RoboDK station: Stringer B Corner-Top-Short-BOX1.rdk

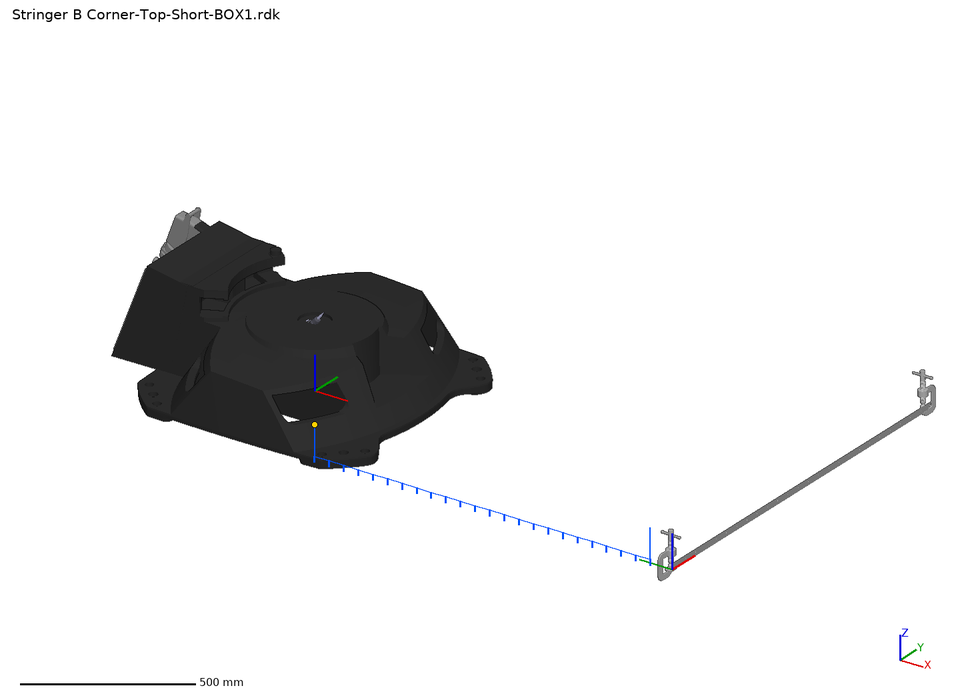
[picture v0: the station drawn from its stored meshes, robots at their saved joint values, targets as dots, program paths as lines]
Station Stringer B Corner-Top-Short-BOX1 (saved by RoboDK 5.2.3). Poses are relative to the parent item; angles as X-Y-Z fixed-axis rotations.
  - frame KUKA KR 210 R2700 extra Base at (0, 0, 0) mm
    - robot KUKA KR 210 R2700 extra: 6 axes, payload 210 kg, reach 2696 mm, repeatability 0.06 mm, weight 1068 kg
        joint limits [-185, -140, -120, -350, -125, -350] to [185, -5, 155, 350, 125, 350]; home [0, -90, 90, 0, 0, 0]; saved at [19.623, -62.154, 124.175, 233.066, 15.332, -216.577]
      - tool Spindle, TCP at (32, 0, 260) mm, rotated rx 0 ry 39 rz 0 deg, size 157.3 x 72 x 259.9 mm
  - frame Frame 2 at (1618.38, -541.41, 103.58) mm, rotated rx 0 ry 0 rz 90 deg
    - object L-Stringer B-top-corner at (0, 0, 0) mm, size 1281.1 x 20 x 20 mm, geometry from L-Stringer B-top-corner.stl
    - object Stringer B Corner-Top-Short-Box1 at (0, 0, 0) mm, rotated rx 0 ry 0 rz -90 deg, 24 curves, geometry from Point 24
  - machining project Point settings: rotZ(0) | rotX(0)*rotY(0) | rotz(0) | onStart | onPathStart | onApproach | onPoint | onRetract | onFinish | SetRPM(%1) | SetTool(%1) | Extruder(%1) | default | default | OutOnMov(%1) | OutOffMov(%1) | onPathFinish | M_RunCode(%1)
  - program Point (131 instructions, listed below)
  - object FinalClamp at (1606.21, -531.49, 164.11) mm, rotated rx 0 ry 90 rz 177.84 deg, size 145.3 x 71.1 x 72 mm, geometry from FinalClamp.stp
  - object FinalClamp2 at (1603.6, 720.64, 166.88) mm, rotated rx 0 ry 88.95 rz 0 deg, size 145.3 x 71.1 x 72 mm, geometry from FinalClamp.stp
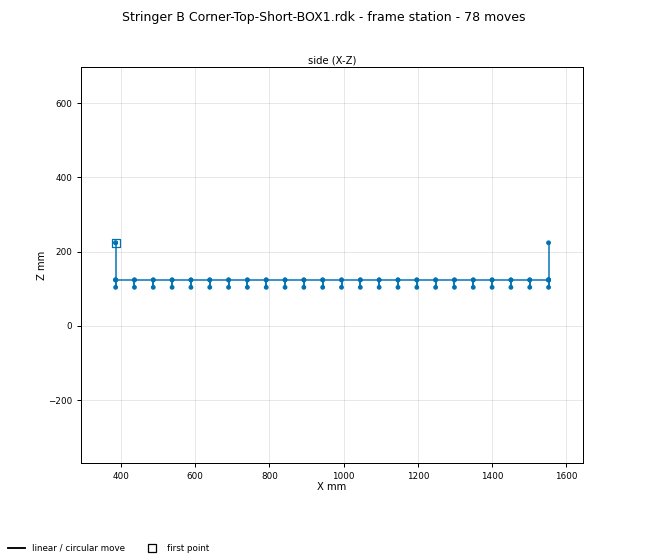
[picture p0: tool path of Stringer B Corner-Top-Short-BOX1.rdk in frame station, 78 of 78 moves have a stored position in this frame; points joined in program order, loops and branches not executed]

--- program Point (robot KUKA KR 210 R2700 extra) ---
  Smooth(1)
  Set speed (1000.0 mm/s)
  Set Ref.: Frame 2
  Set Tool: Spindle
  Show Spindle
  MoveJ 1 to (-12.5, 1232.57, 120) mm, rotated rx 180 ry 0 rz -180 deg; joints [-27.427, -59.782, 119.392, 107.012, 17.647, -129.765]
  MoveL 2 to (-12.5, 1232.57, 120) mm, rotated rx 180 ry 0 rz -180 deg; joints [-27.427, -59.782, 119.392, 107.012, 17.647, -129.765]
  MoveL 3 to (-12.5, 1232.57, 20) mm, rotated rx 180 ry 0 rz -180 deg; joints [-27.427, -54.556, 118.849, 119.827, 19.52, -143.276]
  MoveL 4 to (-12.5, 1232.57, 20) mm, rotated rx 180 ry 0 rz -180 deg; joints [-27.427, -54.556, 118.849, 119.827, 19.52, -143.276]
  Set speed (50.0 mm/s)
  MoveL 5 to (-12.5, 1232.57, 0) mm, rotated rx 180 ry 0 rz -180 deg; joints [-27.427, -53.491, 118.683, 121.974, 19.982, -145.557]
  MoveL 6 to (-12.5, 1232.57, 20) mm, rotated rx 180 ry 0 rz -180 deg; joints [-27.427, -54.556, 118.849, 119.827, 19.52, -143.276]
  Set speed (1000.0 mm/s)
  MoveL 7 to (-12.5, 1181.88, 20) mm, rotated rx -180 ry 0 rz -180 deg; joints [-25.683, -55.081, 120.104, 124.287, 19.275, -146.333]
  Set speed (50.0 mm/s)
  MoveL 8 to (-12.5, 1181.88, 0) mm, rotated rx 180 ry 0 rz -180 deg; joints [-25.683, -53.996, 119.936, 126.394, 19.805, -148.568]
  MoveL 9 to (-12.5, 1181.88, 20) mm, rotated rx -180 ry 0 rz -180 deg; joints [-25.683, -55.081, 120.104, 124.287, 19.275, -146.333]
  Set speed (1000.0 mm/s)
  MoveL 10 to (-12.5, 1131.18, 20) mm, rotated rx 180 ry 0 rz 180 deg; joints [-23.885, -55.566, 121.275, 128.787, 19.081, -149.367]
  Set speed (50.0 mm/s)
  MoveL 11 to (-12.5, 1131.18, 0) mm, rotated rx -180 ry 0 rz -180 deg; joints [-23.885, -54.461, 121.104, 130.827, 19.679, -151.529]
  MoveL 12 to (-12.5, 1131.18, 20) mm, rotated rx 180 ry 0 rz 180 deg; joints [-23.885, -55.566, 121.275, 128.787, 19.081, -149.367]
  Set speed (1000.0 mm/s)
  MoveL 13 to (-12.5, 1080.49, 20) mm, rotated rx -180 ry 0 rz -180 deg; joints [-22.036, -56.01, 122.357, 133.306, 18.934, -152.36]
  Set speed (50.0 mm/s)
  MoveL 14 to (-12.5, 1080.49, 0) mm, rotated rx -180 ry 0 rz -180 deg; joints [-22.036, -54.887, 122.184, 135.253, 19.597, -154.423]
  MoveL 15 to (-12.5, 1080.49, 20) mm, rotated rx -180 ry 0 rz -180 deg; joints [-22.036, -56.01, 122.357, 133.306, 18.934, -152.36]
  Set speed (1000.0 mm/s)
  MoveL 16 to (-12.5, 1029.79, 20) mm, rotated rx -180 ry 0 rz -180 deg; joints [-20.138, -56.414, 123.351, 137.828, 18.828, -155.297]
  Set speed (50.0 mm/s)
  MoveL 17 to (-12.5, 1029.79, 0) mm, rotated rx -180 ry 0 rz -180 deg; joints [-20.138, -55.273, 123.176, 139.659, 19.554, -157.236]
  MoveL 18 to (-12.5, 1029.79, 20) mm, rotated rx -180 ry 0 rz -180 deg; joints [-20.138, -56.414, 123.351, 137.828, 18.828, -155.297]
  Set speed (1000.0 mm/s)
  MoveL 19 to (-12.5, 979.09, 20) mm, rotated rx -180 ry 0 rz -180 deg; joints [-18.192, -56.778, 124.253, 142.337, 18.757, -158.165]
  Set speed (50.0 mm/s)
  MoveL 20 to (-12.5, 979.09, 0) mm, rotated rx -180 ry 0 rz -180 deg; joints [-18.192, -55.619, 124.077, 144.031, 19.543, -159.959]
  MoveL 21 to (-12.5, 979.09, 20) mm, rotated rx -180 ry 0 rz -180 deg; joints [-18.192, -56.778, 124.253, 142.337, 18.757, -158.165]
  Set speed (1000.0 mm/s)
  MoveL 22 to (-12.5, 928.4, 20) mm, rotated rx -180 ry 0 rz -180 deg; joints [-16.202, -57.101, 125.063, 146.822, 18.716, -160.956]
  Set speed (50.0 mm/s)
  MoveL 23 to (-12.5, 928.4, 0) mm, rotated rx 180 ry 0 rz 180 deg; joints [-16.202, -55.926, 124.884, 148.36, 19.557, -162.584]
  MoveL 24 to (-12.5, 928.4, 20) mm, rotated rx -180 ry 0 rz -180 deg; joints [-16.202, -57.101, 125.063, 146.822, 18.716, -160.956]
  Set speed (1000.0 mm/s)
  MoveL 25 to (-12.5, 877.7, 20) mm, rotated rx 180 ry 0 rz 180 deg; joints [-14.171, -57.384, 125.777, 151.275, 18.698, -163.668]
  Set speed (50.0 mm/s)
  MoveL 26 to (-12.5, 877.7, 0) mm, rotated rx 180 ry 0 rz -180 deg; joints [-14.171, -56.195, 125.597, 152.641, 19.588, -165.113]
  MoveL 27 to (-12.5, 877.7, 20) mm, rotated rx 180 ry 0 rz 180 deg; joints [-14.171, -57.384, 125.777, 151.275, 18.698, -163.668]
  Set speed (1000.0 mm/s)
  MoveL 28 to (-12.5, 827.01, 20) mm, rotated rx 180 ry 0 rz -180 deg; joints [-12.103, -57.627, 126.395, 155.692, 18.696, -166.298]
  Set speed (50.0 mm/s)
  MoveL 29 to (-12.5, 827.01, 0) mm, rotated rx 180 ry 0 rz 180 deg; joints [-12.103, -56.425, 126.213, 156.872, 19.63, -167.547]
  MoveL 30 to (-12.5, 827.01, 20) mm, rotated rx 180 ry 0 rz -180 deg; joints [-12.103, -57.627, 126.395, 155.692, 18.696, -166.298]
  Set speed (1000.0 mm/s)
  MoveL 31 to (-12.5, 776.31, 20) mm, rotated rx 180 ry 0 rz 180 deg; joints [-10.002, -57.83, 126.915, 160.072, 18.705, -168.852]
  Set speed (50.0 mm/s)
  MoveL 32 to (-12.5, 776.31, 0) mm, rotated rx -180 ry 0 rz -180 deg; joints [-10.002, -56.617, 126.732, 161.056, 19.676, -169.894]
  MoveL 33 to (-12.5, 776.31, 20) mm, rotated rx 180 ry 0 rz 180 deg; joints [-10.002, -57.83, 126.915, 160.072, 18.705, -168.852]
  Set speed (1000.0 mm/s)
  MoveL 34 to (-12.5, 725.62, 20) mm, rotated rx 180 ry 0 rz 180 deg; joints [-7.875, -57.993, 127.336, 164.416, 18.72, -171.339]
  Set speed (50.0 mm/s)
  MoveL 35 to (-12.5, 725.62, 0) mm, rotated rx -180 ry 0 rz -180 deg; joints [-7.875, -56.771, 127.151, 165.196, 19.721, -172.164]
  MoveL 36 to (-12.5, 725.62, 20) mm, rotated rx 180 ry 0 rz 180 deg; joints [-7.875, -57.993, 127.336, 164.416, 18.72, -171.339]
  Set speed (1000.0 mm/s)
  MoveL 37 to (-12.5, 674.92, 20) mm, rotated rx 180 ry 0 rz -180 deg; joints [-5.724, -58.117, 127.656, 168.731, 18.736, -173.768]
  Set speed (50.0 mm/s)
  MoveL 38 to (-12.5, 674.92, 0) mm, rotated rx -180 ry 0 rz -180 deg; joints [-5.724, -56.888, 127.47, 169.3, 19.76, -174.371]
  MoveL 39 to (-12.5, 674.92, 20) mm, rotated rx 180 ry 0 rz -180 deg; joints [-5.724, -58.117, 127.656, 168.731, 18.736, -173.768]
  Set speed (1000.0 mm/s)
  MoveL 40 to (-12.5, 624.22, 20) mm, rotated rx -180 ry 0 rz -180 deg; joints [-3.558, -58.201, 127.874, 173.021, 18.749, -176.155]
  Set speed (50.0 mm/s)
  MoveL 41 to (-12.5, 624.22, 0) mm, rotated rx 180 ry 0 rz -180 deg; joints [-3.558, -56.967, 127.688, 173.376, 19.789, -176.53]
  MoveL 42 to (-12.5, 624.22, 20) mm, rotated rx -180 ry 0 rz -180 deg; joints [-3.558, -58.201, 127.874, 173.021, 18.749, -176.155]
  Set speed (1000.0 mm/s)
  MoveL 43 to (-12.5, 573.53, 20) mm, rotated rx 180 ry 0 rz -180 deg; joints [-1.381, -58.245, 127.99, 177.296, 18.756, -178.513]
  Set speed (50.0 mm/s)
  MoveL 44 to (-12.5, 573.53, 0) mm, rotated rx 180 ry 0 rz -180 deg; joints [-1.381, -57.009, 127.804, 177.434, 19.805, -178.659]
  MoveL 45 to (-12.5, 573.53, 20) mm, rotated rx 180 ry 0 rz -180 deg; joints [-1.381, -58.245, 127.99, 177.296, 18.756, -178.513]
  Set speed (1000.0 mm/s)
  MoveL 46 to (-12.5, 522.83, 20) mm, rotated rx 180 ry 0 rz 180 deg; joints [0.799, -58.25, 128.004, 181.565, 18.757, -180.86]
  Set speed (50.0 mm/s)
  MoveL 47 to (-12.5, 522.83, 0) mm, rotated rx 180 ry 0 rz 180 deg; joints [0.799, -57.014, 127.818, 181.485, 19.807, -180.776]
  MoveL 48 to (-12.5, 522.83, 20) mm, rotated rx 180 ry 0 rz 180 deg; joints [0.799, -58.25, 128.004, 181.565, 18.757, -180.86]
  Set speed (1000.0 mm/s)
  MoveL 49 to (-12.5, 472.14, 20) mm, rotated rx -180 ry 0 rz -180 deg; joints [2.978, -58.216, 127.915, 185.837, 18.751, -183.214]
  Set speed (50.0 mm/s)
  MoveL 50 to (-12.5, 472.14, 0) mm, rotated rx 180 ry 0 rz 180 deg; joints [2.978, -56.982, 127.729, 185.539, 19.795, -182.899]
  MoveL 51 to (-12.5, 472.14, 20) mm, rotated rx -180 ry 0 rz -180 deg; joints [2.978, -58.216, 127.915, 185.837, 18.751, -183.214]
  Set speed (1000.0 mm/s)
  MoveL 52 to (-12.5, 421.44, 20) mm, rotated rx 180 ry 0 rz 180 deg; joints [5.148, -58.143, 127.724, 190.122, 18.74, -185.591]
  Set speed (50.0 mm/s)
  MoveL 53 to (-12.5, 421.44, 0) mm, rotated rx 180 ry 0 rz 180 deg; joints [5.148, -56.913, 127.538, 189.61, 19.769, -185.048]
  MoveL 54 to (-12.5, 421.44, 20) mm, rotated rx 180 ry 0 rz 180 deg; joints [5.148, -58.143, 127.724, 190.122, 18.74, -185.591]
  Set speed (1000.0 mm/s)
  MoveL 55 to (-12.5, 370.75, 20) mm, rotated rx 180 ry 0 rz 180 deg; joints [7.302, -58.03, 127.431, 194.429, 18.724, -188.007]
  Set speed (50.0 mm/s)
  MoveL 56 to (-12.5, 370.75, 0) mm, rotated rx 180 ry 0 rz 180 deg; joints [7.302, -56.806, 127.246, 193.705, 19.732, -187.241]
  MoveL 57 to (-12.5, 370.75, 20) mm, rotated rx 180 ry 0 rz 180 deg; joints [7.302, -58.03, 127.431, 194.429, 18.724, -188.007]
  Set speed (1000.0 mm/s)
  MoveL 58 to (-12.5, 320.05, 20) mm, rotated rx -180 ry 0 rz 180 deg; joints [9.437, -57.877, 127.037, 198.765, 18.709, -190.478]
  Set speed (50.0 mm/s)
  MoveL 59 to (-12.5, 320.05, 0) mm, rotated rx -180 ry 0 rz -180 deg; joints [9.437, -56.662, 126.854, 197.835, 19.689, -189.493]
  MoveL 60 to (-12.5, 320.05, 20) mm, rotated rx -180 ry 0 rz 180 deg; joints [9.437, -57.877, 127.037, 198.765, 18.709, -190.478]
  Set speed (1000.0 mm/s)
  MoveL 61 to (-12.5, 269.35, 20) mm, rotated rx 180 ry 0 rz 180 deg; joints [11.546, -57.685, 126.544, 203.135, 18.698, -193.013]
  Set speed (50.0 mm/s)
  MoveL 62 to (-12.5, 269.35, 0) mm, rotated rx 180 ry 0 rz 180 deg; joints [11.546, -56.48, 126.361, 202.007, 19.642, -191.818]
  MoveL 63 to (-12.5, 269.35, 20) mm, rotated rx 180 ry 0 rz 180 deg; joints [11.546, -57.685, 126.544, 203.135, 18.698, -193.013]
  Set speed (1000.0 mm/s)
  MoveL 64 to (-12.5, 218.66, 20) mm, rotated rx 180 ry 0 rz -180 deg; joints [13.623, -57.453, 125.952, 207.542, 18.696, -195.623]
  Set speed (50.0 mm/s)
  MoveL 65 to (-12.5, 218.66, 0) mm, rotated rx -180 ry 0 rz -180 deg; joints [13.623, -56.26, 125.771, 206.225, 19.598, -194.228]
  MoveL 66 to (-12.5, 218.66, 20) mm, rotated rx 180 ry 0 rz -180 deg; joints [13.623, -57.453, 125.952, 207.542, 18.696, -195.623]
  Set speed (1000.0 mm/s)
  MoveL 67 to (-12.5, 167.96, 20) mm, rotated rx 180 ry 0 rz 180 deg; joints [15.664, -57.18, 125.263, 211.986, 18.709, -198.312]
  Set speed (50.0 mm/s)
  MoveL 68 to (-12.5, 167.96, 0) mm, rotated rx 180 ry 0 rz 180 deg; joints [15.664, -56.002, 125.084, 210.493, 19.564, -196.731]
  MoveL 69 to (-12.5, 167.96, 20) mm, rotated rx 180 ry 0 rz 180 deg; joints [15.664, -57.18, 125.263, 211.986, 18.709, -198.312]
  Set speed (1000.0 mm/s)
  MoveL 70 to (-12.5, 117.27, 20) mm, rotated rx -180 ry 0 rz -180 deg; joints [17.665, -56.868, 124.479, 216.463, 18.744, -201.082]
  Set speed (50.0 mm/s)
  MoveL 71 to (-12.5, 117.27, 0) mm, rotated rx 180 ry 0 rz 180 deg; joints [17.665, -55.705, 124.301, 214.809, 19.545, -199.331]
  MoveL 72 to (-12.5, 117.27, 20) mm, rotated rx -180 ry 0 rz -180 deg; joints [17.665, -56.868, 124.479, 216.463, 18.744, -201.082]
  Set speed (1000.0 mm/s)
  MoveL 73 to (-12.5, 66.57, 20) mm, rotated rx 180 ry 0 rz 180 deg; joints [19.623, -56.515, 123.601, 220.967, 18.806, -203.931]
  Set speed (50.0 mm/s)
  MoveL 74 to (-12.5, 66.57, 0) mm, rotated rx 180 ry 0 rz 180 deg; joints [19.623, -55.369, 123.425, 219.17, 19.549, -202.028]
  MoveL 75 to (-12.5, 66.57, 20) mm, rotated rx 180 ry 0 rz 180 deg; joints [19.623, -56.515, 123.601, 220.967, 18.806, -203.931]
  MoveL 76 to (-12.5, 66.57, 20) mm, rotated rx 180 ry 0 rz 180 deg; joints [19.623, -56.515, 123.601, 220.967, 18.806, -203.931]
  Set speed (1000.0 mm/s)
  MoveL 77 to (-12.5, 66.57, 20) mm, rotated rx 180 ry 0 rz 180 deg; joints [19.623, -56.515, 123.601, 220.967, 18.806, -203.931]
  MoveL 78 to (-12.5, 66.57, 120) mm, rotated rx 180 ry 0 rz -180 deg; joints [19.623, -62.154, 124.175, 233.066, 15.332, -216.577]
